# EPICS substitutions: vacuum/MAIN_TRUNK/db/su12_agilent4uhv.substitutions
# Agilent4UHV substitutions file

file db/agilent4uhv.db
{
     pattern {LOCA,			DEV,		PORT,		ADDR,	TIMEOUT}
     		 {SU1,			SU1213_1,		4uhv_1,		0,		0.2}
     		 {SU1,			SU1213_2,		4uhv_2,		0,		0.2}
}
file db/agilent4uhv_alias.db
{
     pattern {LOCA,			DEV,		SUB1,					SUB2,					SUB3,						SUB4,				PORT,	ADDR,	TIMEOUT}
     		 {SU1,			SU1213_1,	VU408:IP01:SIP20,		VU409:IP01:SIP20,		VU410:IP01:SIP20,			VU411:IP01:SIP20,	4uhv_1,	0,		0.2}
     		 {SU1,			SU1213_2,	VU412:IP01:SIP20,		VEPU1:IP01:SIP20,		VEPU2:IP01:SIP20,			Empty,		4uhv_2,	0,		0.2}
}
